// TIA Portal V20 export
FUNCTION_BLOCK "FB_MCPManagement"   // FB421, SCL
{ S7_Optimized_Access := 'TRUE' }
// stored: AutoNumber false, MemoryReserve 100, SetENOAutomatically false
   VAR
      sRT_SingleBlock : R_TRIG;
      sSelectionAxe01Jog { S7_SetPoint := 'True'} : Bool;
      sSelectionAxe02Jog { S7_SetPoint := 'True'} : Bool;
      sSelectionAxe03Jog : Bool;
      sSelectionAxe04Jog : Bool;
      sSelectionAxe05Jog : Bool;
      sSelectionAxe06Jog : Bool;
      sSelectionAxe07Jog : Bool;
      sSelectionAxe08Jog : Bool;
      sSelectionAxe09Jog : Bool;
      sSelectionAxe10Jog : Bool;
      sSelectionAxe11Jog : Bool;
      sSelectionAxe12Jog : Bool;
      sSelectionAxe13Jog : Bool;
      sSelectionAxe14Jog : Bool;
      sSelectionAxe15Jog : Bool;
      sSelectionAxe16Jog : Bool;
      sSelectionAxe17Jog : Bool;
      sResetProgramEnmodeRef : Bool;
      sRT_McsWcs { S7_SetPoint := 'True'} : R_TRIG;
      sMemoFeedDisable { S7_SetPoint := 'True'} : Bool;
      sTONChanRef { S7_SetPoint := 'True'} : TON_TIME;
      sFP_TONChanRef { S7_SetPoint := 'True'} : R_TRIG;
   END_VAR
   VAR_TEMP
      tFeedrate : Byte;
      tStartTimerChanRef : Bool;
   END_VAR
BEGIN
   REGION Description header 
       //==================================================================================
       // POSALUX Swiss SA / (C) Copyright 2024
       //----------------------------------------------------------------------------------
       // Title: Management of the general MCP button functionalities
       // Comment/Function: 
       // Author: Gowsigan SRITHARAN
       // Engineering: TIA Portal v17
       //----------------------------------------------------------------------------------
       // Change log table:
       // Version  | Date     | Expert in charge | Changes applied
       // ---------|----------|------------------|------------------------------------
       // 00.00.01 | 20250411 | GSR              | First released version
       // 00.00.02 | 20251010 | WFA              | Femto 5a adaptation
       // ==================================================================================
   END_REGION

   REGION Call Mcp keyboard signals management
       "DB_McpKeyboardSignals"();
   END_REGION

   REGION General MCP buttons
       // JOG
       "LBP_ModeGroup".A_JOG := "MCP1_In".jog;
       "MCP1_Out".LEDjog := "LBP_ModeGroup".E_JOG;

       // MDA
       "LBP_ModeGroup".A_MDA := "MCP1_In".mda;
       "MCP1_Out".LEDmda := "LBP_ModeGroup".E_MDA;

       // AUTO
       "LBP_ModeGroup".A_AUTO := "MCP1_In".auto;
       "MCP1_Out".LEDauto := "LBP_ModeGroup".E_AUTO;

       // INC1
       "LBP_ModeGroup".A_INC1 := "MCP1_In".inc1 AND "LBP_ModeGroup".E_JOG;
       "MCP1_Out".LEDinc1 := "LBP_ModeGroup".E_INC1;

       // INC10
       "LBP_ModeGroup".A_INC10 := "MCP1_In".inc10 AND "LBP_ModeGroup".E_JOG;
       "MCP1_Out".LEDinc10 := "LBP_ModeGroup".E_INC10;

       // INC100
       "LBP_ModeGroup".A_INC100 := "MCP1_In".inc100 AND "LBP_ModeGroup".E_JOG;
       "MCP1_Out".LEDinc100 := "LBP_ModeGroup".E_INC100;

       // INC1000
       "LBP_ModeGroup".A_INC1000 := "MCP1_In".inc1000 AND "LBP_ModeGroup".E_JOG;
       "MCP1_Out".LEDinc1000 := "LBP_ModeGroup".E_INC1000;

       // INC10000
       "LBP_ModeGroup".A_INC10000 := "MCP1_In".inc10000 AND "LBP_ModeGroup".E_JOG;
       "MCP1_Out".LEDinc10000 := "LBP_ModeGroup".E_INC10000;

       // INCVAR
       "LBP_ModeGroup".A_INCVar := "MCP1_In".incVar AND "LBP_ModeGroup".E_JOG;
       "MCP1_Out".LEDincVar := "LBP_ModeGroup".E_INCVar;

       // RESET
       "LBP_Chan1".A_Reset := "MCP1_In".reset;

       // SINGLE BLOCK
       #sRT_SingleBlock(CLK := "MCP1_In".singleBlock);

       IF #sRT_SingleBlock.Q THEN
           "LBP_Chan1".A_SBL := NOT "LBP_Chan1".A_SBL;
       END_IF;

       "MCP1_Out".LEDsingleBlock := "LBP_Chan1".A_SBL;
   END_REGION

   REGION Selection axis in JOG

       // Mode JOG selection axe 01
       IF "MCP1_In".axisX AND "LBP_ModeGroup".E_JOG THEN
           #sSelectionAxe01Jog := TRUE;
           #sSelectionAxe02Jog := FALSE;
           #sSelectionAxe03Jog := FALSE;
           #sSelectionAxe04Jog := FALSE;
           #sSelectionAxe05Jog := FALSE;
           #sSelectionAxe06Jog := FALSE;
           #sSelectionAxe07Jog := FALSE;
           #sSelectionAxe08Jog := FALSE;
           #sSelectionAxe09Jog := FALSE;
       END_IF;

       // Mode JOG selection axe 02
       IF "MCP1_In".axisY AND "LBP_ModeGroup".E_JOG THEN
           #sSelectionAxe01Jog := FALSE;
           #sSelectionAxe02Jog := TRUE;
           #sSelectionAxe03Jog := FALSE;
           #sSelectionAxe04Jog := FALSE;
           #sSelectionAxe05Jog := FALSE;
           #sSelectionAxe06Jog := FALSE;
           #sSelectionAxe07Jog := FALSE;
           #sSelectionAxe08Jog := FALSE;
           #sSelectionAxe09Jog := FALSE;
       END_IF;

       // Mode JOG selection axe 03
       IF "MCP1_In".axisZ AND "LBP_ModeGroup".E_JOG THEN
           #sSelectionAxe01Jog := FALSE;
           #sSelectionAxe02Jog := FALSE;
           #sSelectionAxe03Jog := TRUE;
           #sSelectionAxe04Jog := FALSE;
           #sSelectionAxe05Jog := FALSE;
           #sSelectionAxe06Jog := FALSE;
           #sSelectionAxe07Jog := FALSE;
           #sSelectionAxe08Jog := FALSE;
           #sSelectionAxe09Jog := FALSE;
       END_IF;

       // Mode JOG selection axe 04
       IF "MCP1_In".axis4 AND "LBP_ModeGroup".E_JOG THEN
           #sSelectionAxe01Jog := FALSE;
           #sSelectionAxe02Jog := FALSE;
           #sSelectionAxe03Jog := FALSE;
           #sSelectionAxe04Jog := TRUE;
           #sSelectionAxe05Jog := FALSE;
           #sSelectionAxe06Jog := FALSE;
           #sSelectionAxe07Jog := FALSE;
           #sSelectionAxe08Jog := FALSE;
           #sSelectionAxe09Jog := FALSE;
       END_IF;

       // Mode JOG selection axe 05
       IF "MCP1_In".axis5 AND "LBP_ModeGroup".E_JOG THEN
           #sSelectionAxe01Jog := FALSE;
           #sSelectionAxe02Jog := FALSE;
           #sSelectionAxe03Jog := FALSE;
           #sSelectionAxe04Jog := FALSE;
           #sSelectionAxe05Jog := TRUE;
           #sSelectionAxe06Jog := FALSE;
           #sSelectionAxe07Jog := FALSE;
           #sSelectionAxe08Jog := FALSE;
           #sSelectionAxe09Jog := FALSE;
       END_IF;

       // Mode JOG selection axe 06
       IF "MCP1_In".axis6 AND "LBP_ModeGroup".E_JOG THEN
           #sSelectionAxe01Jog := FALSE;
           #sSelectionAxe02Jog := FALSE;
           #sSelectionAxe03Jog := FALSE;
           #sSelectionAxe04Jog := FALSE;
           #sSelectionAxe05Jog := FALSE;
           #sSelectionAxe06Jog := TRUE;
           #sSelectionAxe07Jog := FALSE;
           #sSelectionAxe08Jog := FALSE;
           #sSelectionAxe09Jog := FALSE;
       END_IF;

       // Mode JOG selection axe 07
       IF "MCP1_In".axis7 AND "LBP_ModeGroup".E_JOG THEN
           #sSelectionAxe01Jog := FALSE;
           #sSelectionAxe02Jog := FALSE;
           #sSelectionAxe03Jog := FALSE;
           #sSelectionAxe04Jog := FALSE;
           #sSelectionAxe05Jog := FALSE;
           #sSelectionAxe06Jog := FALSE;
           #sSelectionAxe07Jog := TRUE;
           #sSelectionAxe08Jog := FALSE;
           #sSelectionAxe09Jog := FALSE;
       END_IF;

       // Mode JOG selection axe 08
       IF "MCP1_In".axis8 AND "LBP_ModeGroup".E_JOG THEN
           #sSelectionAxe01Jog := FALSE;
           #sSelectionAxe02Jog := FALSE;
           #sSelectionAxe03Jog := FALSE;
           #sSelectionAxe04Jog := FALSE;
           #sSelectionAxe05Jog := FALSE;
           #sSelectionAxe06Jog := FALSE;
           #sSelectionAxe07Jog := FALSE;
           #sSelectionAxe08Jog := TRUE;
           #sSelectionAxe09Jog := FALSE;
       END_IF;

       // Mode JOG selection axe 09
       IF "MCP1_In".axis9 AND "LBP_ModeGroup".E_JOG THEN
           #sSelectionAxe01Jog := FALSE;
           #sSelectionAxe02Jog := FALSE;
           #sSelectionAxe03Jog := FALSE;
           #sSelectionAxe04Jog := FALSE;
           #sSelectionAxe05Jog := FALSE;
           #sSelectionAxe06Jog := FALSE;
           #sSelectionAxe07Jog := FALSE;
           #sSelectionAxe08Jog := FALSE;
           #sSelectionAxe09Jog := TRUE;
       END_IF;

       // Reset selection jog
       IF NOT "LBP_ModeGroup".E_JOG THEN
           #sSelectionAxe01Jog := FALSE;
           #sSelectionAxe02Jog := FALSE;
           #sSelectionAxe03Jog := FALSE;
           #sSelectionAxe04Jog := FALSE;
           #sSelectionAxe05Jog := FALSE;
           #sSelectionAxe06Jog := FALSE;
           #sSelectionAxe07Jog := FALSE;
           #sSelectionAxe08Jog := FALSE;
           #sSelectionAxe09Jog := FALSE;
       END_IF;

       // Led Axis
       "MCP1_Out".LEDaxisX := #sSelectionAxe01Jog;
       "MCP1_Out".LEDaxisY := #sSelectionAxe02Jog;
       "MCP1_Out".LEDaxisZ := #sSelectionAxe03Jog;
       "MCP1_Out".LEDaxis4 := #sSelectionAxe04Jog;
       "MCP1_Out".LEDaxis5 := #sSelectionAxe05Jog;
       "MCP1_Out".LEDaxis6 := #sSelectionAxe06Jog;
       "MCP1_Out".LEDaxis7 := #sSelectionAxe07Jog;
       "MCP1_Out".LEDaxis8 := #sSelectionAxe08Jog;
       "MCP1_Out".LEDaxis9 := #sSelectionAxe09Jog;
   END_REGION

   REGION Axis move in JOG
       // Axis 01
       IF #sSelectionAxe01Jog THEN
           "LBP_Axis01_X"."A_Plus" := "MCP1_In".plus;
           "LBP_Axis01_X".A_Minus := "MCP1_In".minus;
           "LBP_Axis01_X".A_RapidTrOR := "MCP1_In".rapidTraverse;
       END_IF;

       // Axis 02
       IF #sSelectionAxe02Jog THEN
           "LBP_Axis02_Y".A_Plus := "MCP1_In".plus;
           "LBP_Axis02_Y".A_Minus := "MCP1_In".minus;
           "LBP_Axis02_Y".A_RapidTrOR := "MCP1_In".rapidTraverse;
       END_IF;

       // Axis 03
       IF #sSelectionAxe03Jog THEN
           "LBP_Axis03_ZM".A_Plus := "MCP1_In".plus;
           "LBP_Axis03_ZM".A_Minus := "MCP1_In".minus;
           "LBP_Axis03_ZM".A_RapidTrOR := "MCP1_In".rapidTraverse;
       END_IF;

       // Axis 04
       IF #sSelectionAxe04Jog THEN
           "LBP_Axis04_B".A_Plus := "MCP1_In".plus;
           "LBP_Axis04_B".A_Minus := "MCP1_In".minus;
           "LBP_Axis04_B".A_RapidTrOR := "MCP1_In".rapidTraverse;
       END_IF;

       // Axis 05
       IF #sSelectionAxe05Jog THEN
           "LBP_Axis05_U1".A_Plus := "MCP1_In".plus;
           "LBP_Axis05_U1".A_Minus := "MCP1_In".minus;
           "LBP_Axis05_U1".A_RapidTrOR := "MCP1_In".rapidTraverse;
       END_IF;

       // Axis 06
       IF #sSelectionAxe06Jog THEN
           "LBP_Axis06_U2".A_Plus := "MCP1_In".plus;
           "LBP_Axis06_U2".A_Minus := "MCP1_In".minus;
           "LBP_Axis06_U2".A_RapidTrOR := "MCP1_In".rapidTraverse;
       END_IF;

       // Axe 07
       IF #sSelectionAxe07Jog THEN
           "LBP_Axis07_V".A_Plus := "MCP1_In".plus;
           "LBP_Axis07_V".A_Minus := "MCP1_In".minus;
           "LBP_Axis07_V".A_RapidTrOR := "MCP1_In".rapidTraverse;
       END_IF;

       // Axis 08
       IF #sSelectionAxe08Jog THEN
           "LBP_Axis08_W".A_Plus := "MCP1_In".plus;
           "LBP_Axis08_W".A_Minus := "MCP1_In".minus;
           "LBP_Axis08_W".A_RapidTrOR := "MCP1_In".rapidTraverse;
       END_IF;

       // Axis 09
       IF #sSelectionAxe09Jog THEN
           "LBP_Axis09_ZL".A_Plus := "MCP1_In".plus;
           "LBP_Axis09_ZL".A_Minus := "MCP1_In".minus;
           "LBP_Axis09_ZL".A_RapidTrOR := "MCP1_In".rapidTraverse;
       END_IF;
   END_REGION

   REGION Start and stop feedrate
   // FeedStart/Stop
   IF (NOT "MCP1_In".feedrateStop) AND (NOT "MCP1_In".feedrateStart) THEN
       #sMemoFeedDisable:= TRUE;
   ELSIF "MCP1_In".feedrateStop AND  "MCP1_In".feedrateStart THEN
       #sMemoFeedDisable:= FALSE;
   END_IF;
   "LBP_Chan1".A_FDdisable := #sMemoFeedDisable;

   // LED FeedStop
   "MCP1_Out".LEDfeedrateStop := #sMemoFeedDisable;
   "MCP1_Out".LEDfeedrateStart := NOT #sMemoFeedDisable;
   END_REGION

   REGION Channel feedrate override
       // Activation de la correction de l'avance
       "LBP_Chan1".A_FD_ORA := TRUE;

       #tFeedrate.%X0 := "MCP1_In".feedrateOvrA;
       #tFeedrate.%X1 := "MCP1_In".feedrateOvrB;
       #tFeedrate.%X2 := "MCP1_In".feedrateOvrC;
       #tFeedrate.%X3 := "MCP1_In".feedrateOvrD;
       #tFeedrate.%X4 := "MCP1_In".feedrateOvrE;
       #tFeedrate.%X5 := FALSE;
       #tFeedrate.%X6 := FALSE;
       #tFeedrate.%X7 := FALSE;

       // Forcing the override at 100% between 20% and 120% in manual/MDA mode WFA A REVOIR
       // IF NOT "LBP_ModeGroup".E_JOG AND #tFeedrate >= 8 THEN
       //     "LBP_Chan1".A_FD_OR := 26;
       // ELSE
           "LBP_Chan1".A_FD_OR     := #tFeedrate;
           "LBP_Axis01_X".A_FD_OR  := #tFeedrate;
           "LBP_Axis02_Y".A_FD_OR  := #tFeedrate;
           "LBP_Axis03_ZM".A_FD_OR := #tFeedrate;
           "LBP_Axis04_B".A_FD_OR  := #tFeedrate;
           "LBP_Axis05_U1".A_FD_OR := #tFeedrate;
           "LBP_Axis06_U2".A_FD_OR := #tFeedrate;
           "LBP_Axis07_V".A_FD_OR  := #tFeedrate;
           "LBP_Axis08_W".A_FD_OR  := #tFeedrate;
           "LBP_Axis09_ZL".A_FD_OR := #tFeedrate;
       // END_IF;
   END_REGION

   REGION Axis override
       // Allows modifying the movement speed OF the axis using the feed potentiometer
       "LBP_Axis01_X".A_ORactive  := TRUE;
       "LBP_Axis02_Y".A_ORactive  := TRUE;
       "LBP_Axis03_ZM".A_ORactive := TRUE;
       "LBP_Axis04_B".A_ORactive  := TRUE;
       "LBP_Axis05_U1".A_ORactive := TRUE;
       "LBP_Axis06_U2".A_ORactive := TRUE;
       "LBP_Axis07_V".A_ORactive  := TRUE;
       "LBP_Axis08_W".A_ORactive  := TRUE;
       "LBP_Axis09_ZL".A_ORactive := TRUE;
   END_REGION

   REGION Rapid traverse override active
       // Allows adjustment of the axis movement speed using the feed potentiometer
       "LBP_Chan1".A_RT_ORA := TRUE;
       "LBP_Chan1".A_RT_OR := "LBP_Chan1".A_FD_OR;
   END_REGION

   REGION Switching between MCS and WCS
       #sRT_McsWcs(CLK := "MCP1_In".mcsWcs OR  "LBP_HMI".E_ActWCS);
       IF #sRT_McsWcs.Q THEN
           "LBP_HMI".A_ActWCS := NOT "LBP_HMI".A_ActWCS;
       END_IF;
       "MCP1_Out".LEDmcsWcs := NOT "LBP_HMI".A_ActWCS;
   END_REGION

   REGION Key Switch signals
       "LBP_NC".A_Keyswitch0 := "MCP1_In".keySwitch0;
       "LBP_NC".A_Keyswitch1 := "MCP1_In".keySwitch1;
       "LBP_NC".A_Keyswitch2 := "MCP1_In".keySwitch2;
       "LBP_NC".A_Keyswitch3 := "MCP1_In".keySwitch3;
   END_REGION

   REGION Channel Referencing
       "LBP_ModeGroup".A_REF := "MCP1_In".refPoint;

       IF ("LBP_ModeGroup".E_REF
           AND NOT "LBP_Chan1".A_Ref)
           OR ("LBP_ModeGroup".E_REF
           AND "LBP_Chan1".A_Ref
           AND "Clock_1.25Hz") THEN
           "MCP1_Out".LEDrefPoint := TRUE;
       ELSE
           "MCP1_Out".LEDrefPoint := FALSE;
       END_IF;

       IF "LBP_ModeGroup".E_JOG
           AND "LBP_ModeGroup".E_REF
           AND "LBP_Chan1".A_NCStart THEN
           "LBP_Chan1".A_Ref := TRUE;
       END_IF;

       #tStartTimerChanRef :=
       "LBP_Chan1".E_AxesRef
       AND NOT "LBP_Chan1".E_Ref
       AND "LBP_Chan1".A_Ref
       AND "LBP_Chan1".E_ChanReset;

       #sTONChanRef(IN := #tStartTimerChanRef,
                    PT := T#500MS);

       #sFP_TONChanRef(CLK := #sTONChanRef.Q);

       IF #sFP_TONChanRef.Q THEN
           "LBP_ModeGroup".A_JOG := TRUE;
       END_IF;

       IF #sFP_TONChanRef.Q OR "LBP_Chan1".A_Reset THEN
           "LBP_Chan1".A_Ref := FALSE;
       END_IF;
   END_REGION

   REGION Reset group mode
       "LBP_ModeGroup".A_MGReset := "LBP_NC".E_NCKalarm AND "LBP_Chan1".A_Reset;
   END_REGION
END_FUNCTION_BLOCK
